(* CODESYS project vestidor.project
   Title: pl3
   Version: 0.0.0.0
   Author: ALUMNO

Project tree, tasks and I/O mapping:
  MyController : TM241CEC24R, Schneider Electric, order no. TM241CEC24R, version 4.0.6.18
      settings: OPCUA enable = True; Dummy int param for online change = 17
    application Application
      task MAST (cyclic, interval 20 ms, priority 15, watchdog 100 ms x 1) calls Main
      global variables GVL
      program Ua_control [FBD]
      OPCUASymbolConfiguration
      program Main [FBD]
      program Local_control [FBD]
    DI : Digital Inputs, Schneider Electric, version 4.0.6.18
        input  iwDI_IW0 : WORD  // IW0
        input  Application.Local_control.boolResetLocal : BOOL  // IW0.I0
        input  Application.Main.boolDeactivateStop : BOOL  // IW0.I1
        input  Application.Local_control.boolSetPosition : BOOL  // IW0.I2
        input  ibDI_IB1 : BYTE  // IB1
    DQ : Digital Outputs, Schneider Electric, version 4.0.6.18
        output Application.Main.ledLocalControl : BOOL  // QW0.Q0
        output Application.Main.ledUaControl : BOOL  // QW0.Q1
        output qbDQ_QB1 : BYTE  // QB1
        unmapped channels: QW0
    Counters : Counters, Schneider Electric, version 4.0.6.18
    Pulse_Generators : Pulse Generators, Schneider Electric, version 4.0.6.18
    Cartridge_1 : Cartridge, Schneider Electric, version 4.0.6.18
    IO_Bus : IO bus - TM3, Schneider Electric, version 4.0.6.18
    COM_Bus : COM bus, Schneider Electric, version 4.0.6.18
    Ethernet_1 : Ethernet Network, Schneider Electric, version 4.0.6.18
        settings: IPAddress = [10, 0, 0, 41]; SubnetMask = [255, 255, 0, 0]; GatewayAddress = [10, 0, 0, 1]; WebServer = TRUE; FTP Server = TRUE; SoMachine Protocol = TRUE; Modbus Server = TRUE; NetManage Protocol = TRUE; SNMP protocol = TRUE; Enable Routing = FALSE; WebVisu protocol = TRUE; DHCP Server Active = TRUE
    Serial_Line_1 : Serial line, Schneider Electric, version 4.0.6.18
      SoMachine_Network_Manager : SoMachine-Network Manager, Schneider Electric, version 4.0.0.2
    Serial_Line_2 : Serial line, Schneider Electric, version 4.0.6.18
      Modbus_Manager : Modbus Manager, Schneider Electric, version 4.0.0.2
    CAN_1 : CANopen bus, Schneider Electric, version 4.0.6.18
      CANopen_Performance : CANopen Performance, Schneider Electric, order no. 1806, version 3.0.1.24
          settings: ConfigVersion = 50659584
        Lexium_32_M : Lexium 32 M, Schneider Electric, order no. 91200, version 3.5.9.0
            settings: General Options.Optional Device = TRUE; NODEIDSAVED = 1; SDO Timeout = 1000000; Explicit Deactivate PDOs = FALSE; EXPERTSETTINGS = True; Heartbeat-Producer Time = 200; PDO 16#1400.COBID = 16#0201; PDO 16#1801.COBID = 16#C0000281; Generic COBID = '$NODEID+16#C0000280'; PDO 16#1802.COBID = 16#C0000381; Generic COBID = '$NODEID+16#C0000380'; PDO 16#1803.COBID = 16#40000481; Generic COBID = '$NODEID+16#C0000480'; Heartbeat-Consuming1.Heartbeat-Time = 300 ms; Controlword.Subindex = 16#00; Target position.Subindex = 16#00; Controlword.Subindex = 16#00; Target velocity.Subindex = 16#00; Statusword.Subindex = 16#00; Position actual value.Subindex = 16#00; Statusword.Subindex = 16#00; Velocity actual value.Subindex = 16#00; _IO_act.Index = 16#3008; _IO_act.Subindex = 16#01; _IO_act.ObjectLength = 16; _IOM1_AI11_act.Index = 16#304F; _IOM1_AI11_act.Subindex = 16#01; _IOM1_AI11_act.ObjectLength = 16; SDO List.Set Guardtime.Index = 16#100C; SDO List.Set Guardtime.Subindex = 16#00; SDO List.Set Guardtime.Value = 16#00000000; SDO List.Set Guardtime.Size = 16; SDO List.Set Guardtime.AbortIfError = FALSE; SDO List.Set Guardtime.JumpToLine = FALSE; SDO List.Set Guardtime.Line = 0; SDO List.Set Lifetime.Index = 16#100D; SDO List.Set Lifetime.Subindex = 16#00; SDO List.Set Lifetime.Value = 16#00000000; SDO List.Set Lifetime.Size = 8; SDO List.Set Lifetime.AbortIfError = FALSE;
              SDO List.Set Lifetime.JumpToLine = FALSE; SDO List.Set Lifetime.Line = 0; SDO List.Disable Emcy CobID.Index = 16#1014; SDO List.Disable Emcy CobID.Subindex = 16#00; SDO List.Disable Emcy CobID.Value = 16#80000081; SDO List.Disable Emcy CobID.Size = 32; SDO List.Disable Emcy CobID.AbortIfError = FALSE; SDO List.Disable Emcy CobID.JumpToLine = FALSE; SDO List.Disable Emcy CobID.Line = 0; SDO List.Set Emcy CobID.Index = 16#1014; SDO List.Set Emcy CobID.Subindex = 16#00; SDO List.Set Emcy CobID.Value = 16#00000081; SDO List.Set Emcy CobID.Size = 32; SDO List.Set Emcy CobID.AbortIfError = FALSE; SDO List.Set Emcy CobID.JumpToLine = FALSE; SDO List.Set Emcy CobID.Line = 0; SDO List.Set Heartbeat Consumer.Index = 16#1016; SDO List.Set Heartbeat Consumer.Subindex = 16#01; SDO List.Set Heartbeat Consumer.Value = 16#007F012C; SDO List.Set Heartbeat Consumer.Size = 32; SDO List.Set Heartbeat Consumer.AbortIfError = FALSE; SDO List.Set Heartbeat Consumer.JumpToLine = FALSE; SDO List.Set Heartbeat Consumer.Line = 0; SDO List.Set Heartbeat Consumer.Index = 16#1016; SDO List.Set Heartbeat Consumer.Subindex = 16#02; SDO List.Set Heartbeat Consumer.Value = 0; SDO List.Set Heartbeat Consumer.Size = 32; SDO List.Set Heartbeat Consumer.AbortIfError = FALSE; SDO List.Set Heartbeat Consumer.JumpToLine = FALSE; SDO List.Set Heartbeat Consumer.Line = 0; SDO List.Set Heartbeat Consumer.Index = 16#1016; SDO List.Set Heartbeat Consumer.Subindex = 16#03; SDO List.Set Heartbeat Consumer.Value = 0; SDO List.Set Heartbeat Consumer.Size = 32; SDO List.Set Heartbeat Consumer.AbortIfError = FALSE; SDO List.Set Heartbeat Consumer.JumpToLine = FALSE; SDO List.Set Heartbeat Consumer.Line = 0; SDO List.Set Heartbeat Producer.Index = 16#1017; SDO List.Set Heartbeat Producer.Subindex = 16#00; SDO List.Set Heartbeat Producer.Value = 16#000000C8;
              SDO List.Set Heartbeat Producer.Size = 16; SDO List.Set Heartbeat Producer.AbortIfError = FALSE; SDO List.Set Heartbeat Producer.JumpToLine = FALSE; SDO List.Set Heartbeat Producer.Line = 0; SDO List.Disable PDO.Index = 16#1400; SDO List.Disable PDO.Subindex = 16#01; SDO List.Disable PDO.Value = 16#80000201; SDO List.Disable PDO.Size = 32; SDO List.Disable PDO.AbortIfError = FALSE; SDO List.Disable PDO.JumpToLine = FALSE; SDO List.Disable PDO.Line = 0; SDO List.Set transmission type.Index = 16#1400; SDO List.Set transmission type.Subindex = 16#02; SDO List.Set transmission type.Value = 16#FF; SDO List.Set transmission type.Size = 8; SDO List.Set transmission type.AbortIfError = FALSE; SDO List.Set transmission type.JumpToLine = FALSE; SDO List.Set transmission type.Line = 0; SDO List.Clear pdo mapping.Index = 16#1600; SDO List.Clear pdo mapping.Subindex = 16#00; SDO List.Clear pdo mapping.Value = 16#0; SDO List.Clear pdo mapping.Size = 8; SDO List.Clear pdo mapping.AbortIfError = FALSE; SDO List.Clear pdo mapping.JumpToLine = FALSE; SDO List.Clear pdo mapping.Line = 0; SDO List.Set Mapping.Index = 16#1600; SDO List.Set Mapping.Subindex = 16#01; SDO List.Set Mapping.Value = 16#301B1F10; SDO List.Set Mapping.Size = 32; SDO List.Set Mapping.AbortIfError = FALSE; SDO List.Set Mapping.JumpToLine = FALSE; SDO List.Set Mapping.Line = 0; SDO List.Set Mapping.Index = 16#1600; SDO List.Set Mapping.Subindex = 16#02; SDO List.Set Mapping.Value = 16#301B2210; SDO List.Set Mapping.Size = 32; SDO List.Set Mapping.AbortIfError = FALSE; SDO List.Set Mapping.JumpToLine = FALSE; SDO List.Set Mapping.Line = 0; SDO List.Set Mapping.Index = 16#1600;
              SDO List.Set Mapping.Subindex = 16#03; SDO List.Set Mapping.Value = 16#301B2120; SDO List.Set Mapping.Size = 32; SDO List.Set Mapping.AbortIfError = FALSE; SDO List.Set Mapping.JumpToLine = FALSE; SDO List.Set Mapping.Line = 0; SDO List.Set number of pdos.Index = 16#1600; SDO List.Set number of pdos.Subindex = 16#00; SDO List.Set number of pdos.Value = 16#03; SDO List.Set number of pdos.Size = 8; SDO List.Set number of pdos.AbortIfError = FALSE; SDO List.Set number of pdos.JumpToLine = FALSE; SDO List.Set number of pdos.Line = 0; SDO List.Set and enable COB-ID.Index = 16#1400; SDO List.Set and enable COB-ID.Subindex = 16#01; SDO List.Set and enable COB-ID.Value = 16#00000201; SDO List.Set and enable COB-ID.Size = 32; SDO List.Set and enable COB-ID.AbortIfError = FALSE; SDO List.Set and enable COB-ID.JumpToLine = FALSE; SDO List.Set and enable COB-ID.Line = 0; SDO List.Disable PDO.Index = 16#1401; SDO List.Disable PDO.Subindex = 16#01; SDO List.Disable PDO.Value = 16#80000301; SDO List.Disable PDO.Size = 32; SDO List.Disable PDO.AbortIfError = FALSE; SDO List.Disable PDO.JumpToLine = FALSE; SDO List.Disable PDO.Line = 0; SDO List.Disable PDO.Index = 16#1402; SDO List.Disable PDO.Subindex = 16#01; SDO List.Disable PDO.Value = 16#80000401; SDO List.Disable PDO.Size = 32; SDO List.Disable PDO.AbortIfError = FALSE; SDO List.Disable PDO.JumpToLine = FALSE; SDO List.Disable PDO.Line = 0; SDO List.Disable PDO.Index = 16#1403; SDO List.Disable PDO.Subindex = 16#01; SDO List.Disable PDO.Value = 16#80000501; SDO List.Disable PDO.Size = 32; SDO List.Disable PDO.AbortIfError = FALSE; SDO List.Disable PDO.JumpToLine = FALSE;
              SDO List.Disable PDO.Line = 0; SDO List.Disable PDO.Index = 16#1800; SDO List.Disable PDO.Subindex = 16#01; SDO List.Disable PDO.Value = 16#C0000181; SDO List.Disable PDO.Size = 32; SDO List.Disable PDO.AbortIfError = FALSE; SDO List.Disable PDO.JumpToLine = FALSE; SDO List.Disable PDO.Line = 0; SDO List.Set transmission type.Index = 16#1800; SDO List.Set transmission type.Subindex = 16#02; SDO List.Set transmission type.Value = 16#FF; SDO List.Set transmission type.Size = 8; SDO List.Set transmission type.AbortIfError = FALSE; SDO List.Set transmission type.JumpToLine = FALSE; SDO List.Set transmission type.Line = 0; SDO List.Set inhibit time.Index = 16#1800; SDO List.Set inhibit time.Subindex = 16#03; SDO List.Set inhibit time.Value = 16#0064; SDO List.Set inhibit time.Size = 16; SDO List.Set inhibit time.AbortIfError = FALSE; SDO List.Set inhibit time.JumpToLine = FALSE; SDO List.Set inhibit time.Line = 0; SDO List.Set event time.Index = 16#1800; SDO List.Set event time.Subindex = 16#05; SDO List.Set event time.Value = 16#0000; SDO List.Set event time.Size = 16; SDO List.Set event time.AbortIfError = FALSE; SDO List.Set event time.JumpToLine = FALSE; SDO List.Set event time.Line = 0; SDO List.Clear pdo mapping.Index = 16#1A00; SDO List.Clear pdo mapping.Subindex = 16#00; SDO List.Clear pdo mapping.Value = 16#0; SDO List.Clear pdo mapping.Size = 8; SDO List.Clear pdo mapping.AbortIfError = FALSE; SDO List.Clear pdo mapping.JumpToLine = FALSE; SDO List.Clear pdo mapping.Line = 0; SDO List.Set Mapping.Index = 16#1A00; SDO List.Set Mapping.Subindex = 16#01; SDO List.Set Mapping.Value = 16#301B2510; SDO List.Set Mapping.Size = 32;
              SDO List.Set Mapping.AbortIfError = FALSE; SDO List.Set Mapping.JumpToLine = FALSE; SDO List.Set Mapping.Line = 0; SDO List.Set Mapping.Index = 16#1A00; SDO List.Set Mapping.Subindex = 16#02; SDO List.Set Mapping.Value = 16#301B2610; SDO List.Set Mapping.Size = 32; SDO List.Set Mapping.AbortIfError = FALSE; SDO List.Set Mapping.JumpToLine = FALSE; SDO List.Set Mapping.Line = 0; SDO List.Set Mapping.Index = 16#1A00; SDO List.Set Mapping.Subindex = 16#03; SDO List.Set Mapping.Value = 16#301B2710; SDO List.Set Mapping.Size = 32; SDO List.Set Mapping.AbortIfError = FALSE; SDO List.Set Mapping.JumpToLine = FALSE; SDO List.Set Mapping.Line = 0; SDO List.Set Mapping.Index = 16#1A00; SDO List.Set Mapping.Subindex = 16#04; SDO List.Set Mapping.Value = 16#301B2810; SDO List.Set Mapping.Size = 32; SDO List.Set Mapping.AbortIfError = FALSE; SDO List.Set Mapping.JumpToLine = FALSE; SDO List.Set Mapping.Line = 0; SDO List.Set number of pdos.Index = 16#1A00; SDO List.Set number of pdos.Subindex = 16#00; SDO List.Set number of pdos.Value = 16#04; SDO List.Set number of pdos.Size = 8; SDO List.Set number of pdos.AbortIfError = FALSE; SDO List.Set number of pdos.JumpToLine = FALSE; SDO List.Set number of pdos.Line = 0; SDO List.Set and enable COB-ID.Index = 16#1800; SDO List.Set and enable COB-ID.Subindex = 16#01; SDO List.Set and enable COB-ID.Value = 16#40000181; SDO List.Set and enable COB-ID.Size = 32; SDO List.Set and enable COB-ID.AbortIfError = FALSE; SDO List.Set and enable COB-ID.JumpToLine = FALSE; SDO List.Set and enable COB-ID.Line = 0; SDO List.Disable PDO.Index = 16#1801; SDO List.Disable PDO.Subindex = 16#01;
              SDO List.Disable PDO.Value = 16#C0000281; SDO List.Disable PDO.Size = 32; SDO List.Disable PDO.AbortIfError = FALSE; SDO List.Disable PDO.JumpToLine = FALSE; SDO List.Disable PDO.Line = 0; SDO List.Disable PDO.Index = 16#1802; SDO List.Disable PDO.Subindex = 16#01; SDO List.Disable PDO.Value = 16#C0000381; SDO List.Disable PDO.Size = 32; SDO List.Disable PDO.AbortIfError = FALSE; SDO List.Disable PDO.JumpToLine = FALSE; SDO List.Disable PDO.Line = 0; SDO List.Disable PDO.Index = 16#1803; SDO List.Disable PDO.Subindex = 16#01; SDO List.Disable PDO.Value = 16#C0000481; SDO List.Disable PDO.Size = 32; SDO List.Disable PDO.AbortIfError = FALSE; SDO List.Disable PDO.JumpToLine = FALSE; SDO List.Disable PDO.Line = 0; SDO List.Set transmission type.Index = 16#1803; SDO List.Set transmission type.Subindex = 16#02; SDO List.Set transmission type.Value = 16#FE; SDO List.Set transmission type.Size = 8; SDO List.Set transmission type.AbortIfError = FALSE; SDO List.Set transmission type.JumpToLine = FALSE; SDO List.Set transmission type.Line = 0; SDO List.Set inhibit time.Index = 16#1803; SDO List.Set inhibit time.Subindex = 16#03; SDO List.Set inhibit time.Value = 16#0000; SDO List.Set inhibit time.Size = 16; SDO List.Set inhibit time.AbortIfError = FALSE; SDO List.Set inhibit time.JumpToLine = FALSE; SDO List.Set inhibit time.Line = 0; SDO List.Set event time.Index = 16#1803; SDO List.Set event time.Subindex = 16#05; SDO List.Set event time.Value = 16#0000; SDO List.Set event time.Size = 16; SDO List.Set event time.AbortIfError = FALSE; SDO List.Set event time.JumpToLine = FALSE; SDO List.Set event time.Line = 0;
              SDO List.Clear pdo mapping.Index = 16#1A03; SDO List.Clear pdo mapping.Subindex = 16#00; SDO List.Clear pdo mapping.Value = 16#0; SDO List.Clear pdo mapping.Size = 8; SDO List.Clear pdo mapping.AbortIfError = FALSE; SDO List.Clear pdo mapping.JumpToLine = FALSE; SDO List.Clear pdo mapping.Line = 0; SDO List.Set Mapping.Index = 16#1A03; SDO List.Set Mapping.Subindex = 16#01; SDO List.Set Mapping.Value = 16#30080110; SDO List.Set Mapping.Size = 32; SDO List.Set Mapping.AbortIfError = FALSE; SDO List.Set Mapping.JumpToLine = FALSE; SDO List.Set Mapping.Line = 0; SDO List.Set Mapping.Index = 16#1A03; SDO List.Set Mapping.Subindex = 16#02; SDO List.Set Mapping.Value = 16#304F0110; SDO List.Set Mapping.Size = 32; SDO List.Set Mapping.AbortIfError = FALSE; SDO List.Set Mapping.JumpToLine = FALSE; SDO List.Set Mapping.Line = 0; SDO List.Set number of pdos.Index = 16#1A03; SDO List.Set number of pdos.Subindex = 16#00; SDO List.Set number of pdos.Value = 16#02; SDO List.Set number of pdos.Size = 8; SDO List.Set number of pdos.AbortIfError = FALSE; SDO List.Set number of pdos.JumpToLine = FALSE; SDO List.Set number of pdos.Line = 0; SDO List.Set and enable COB-ID.Index = 16#1803; SDO List.Set and enable COB-ID.Subindex = 16#01; SDO List.Set and enable COB-ID.Value = 16#40000481; SDO List.Set and enable COB-ID.Size = 32; SDO List.Set and enable COB-ID.AbortIfError = FALSE; SDO List.Set and enable COB-ID.JumpToLine = FALSE; SDO List.Set and enable COB-ID.Line = 0; SDO List.Automap SDO1.Index = 16#3041; SDO List.Automap SDO1.Subindex = 16#0B; SDO List.Automap SDO1.Value = 15; SDO List.Automap SDO1.Size = 16; SDO List.Automap SDO1.AbortIfError = FALSE;
              SDO List.Automap SDO1.JumpToLine = FALSE; SDO List.Automap SDO1.Line = 0; SDO List.Automap SDO2.Index = 16#301B; SDO List.Automap SDO2.Subindex = 16#08; SDO List.Automap SDO2.Value = 1; SDO List.Automap SDO2.Size = 16; SDO List.Automap SDO2.AbortIfError = FALSE; SDO List.Automap SDO2.JumpToLine = FALSE; SDO List.Automap SDO2.Line = 0; SDO List.Automap SDO3.Index = 16#301B; SDO List.Automap SDO3.Subindex = 16#1E; SDO List.Automap SDO3.Value = 10; SDO List.Automap SDO3.Size = 16; SDO List.Automap SDO3.AbortIfError = FALSE; SDO List.Automap SDO3.JumpToLine = FALSE; SDO List.Automap SDO3.Line = 0; ConfigVersion = 50659584
            input  Application.Local_control.boolPowerOnLocal : BOOL  // _IO_act.Bit1
            input  Application.Main.isLocal : BOOL  // _IO_act.Bit5
            input  Application.Local_control.potentiometer1 : INT  // _IOM1_AI11_act
            unmapped channels: driveModeCtrl, RefA16, RefB32, driveStat, mfStat, motionStat, driveInput, _IO_act
*)

// MyController/Application/GVL
VAR_GLOBAL
	max_vel: INT:=200;
END_VAR

// MyController/Application/Main
PROGRAM Main
VAR
	//////////////////////
	TORQUE_MAX: INT:= 300;	
	//////////////////////
	
	// Para decidir que POU correr
	isLocal: BOOL; // Asignado a PDO
	// Leds para indicarlo
	ledUaControl: BOOL; // Asginado a DQ del PLC
	ledLocalControl: BOOL; // Asignado a DQ del PLC
	// Para hacer halt en cambio de control local a Ua
	isHalt: BOOL;
	FallingEdgeLocalControl_trigg: F_TRIG;
	HaltStopLocalControlModule: MC_Halt_LXM;
	// Lectura continua del torque para parada de emergencia
	TorqueReadModule: MC_ReadActualTorque_LXM;
	actualTorque: INT;
	boolDeactivateStop: BOOL; // Asignado a DI del PLC
	HighTorqueSetReset: SR;
	isHighTorque: BOOL;
	HighTorqueStopModule: MC_Stop_LXM;	
	isStop: BOOL;
END_VAR
VAR // added by the converter: edge detectors and wires of the graphical bodies
    _w1, _w2 : BOOL;
END_VAR

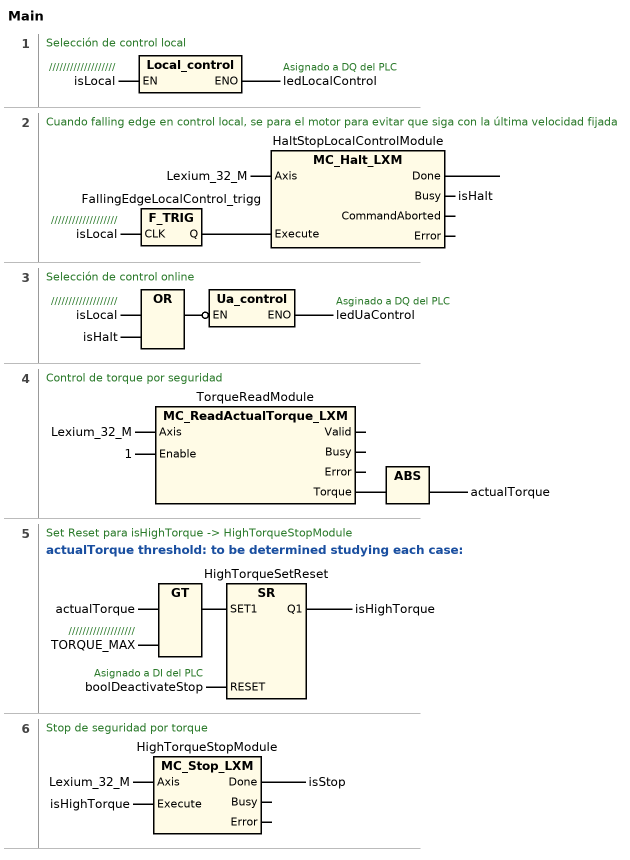
// NETWORK 1
// Selección de control local
//   isLocal: ///////////////////
//   ledLocalControl: Asignado a DQ del PLC
_w1 := isLocal;
IF _w1 THEN Local_control(); END_IF
ledLocalControl := _w1;

// NETWORK 2
// Cuando falling edge en control local, se para el motor para evitar que siga con la última velocidad fijada
//   isLocal: ///////////////////
FallingEdgeLocalControl_trigg(CLK := isLocal); // F_TRIG
HaltStopLocalControlModule(Axis := Lexium_32_M, Execute := FallingEdgeLocalControl_trigg.Q, Busy => isHalt); // MC_Halt_LXM

// NETWORK 3
// Selección de control online
//   isLocal: ///////////////////
//   ledUaControl: Asginado a DQ del PLC
_w2 := NOT (isLocal OR isHalt);
IF _w2 THEN Ua_control(); END_IF
ledUaControl := _w2;

// NETWORK 4
// Control de torque por seguridad
//   TorqueReadModule: Lectura continua del torque para parada de emergencia
TorqueReadModule(Axis := Lexium_32_M, Enable := 1); // MC_ReadActualTorque_LXM
actualTorque := ABS(TorqueReadModule.Torque);

// NETWORK 5
// Set Reset para isHighTorque -> HighTorqueStopModule
//   TORQUE_MAX: ///////////////////
//   boolDeactivateStop: Asignado a DI del PLC
// label: actualTorque threshold: to be determined studying each case
HighTorqueSetReset(SET1 := actualTorque > TORQUE_MAX, RESET := boolDeactivateStop); // SR
isHighTorque := HighTorqueSetReset.Q1;

// NETWORK 6
// Stop de seguridad por torque
HighTorqueStopModule(Axis := Lexium_32_M, Execute := isHighTorque); // MC_Stop_LXM
isStop := HighTorqueStopModule.Done;

END_PROGRAM

// MyController/Application/Local_control
PROGRAM Local_control
VAR
	//////////////////////////
	POT_MAX_VALUE: INT:=10000;
	DEAD_ZONE: INT:=1000;	
	//////////////////////////
	
	boolPowerOnLocal: BOOL;  // Asignado a PDO
	PowerOnModuleLocal: MC_Power_LXM;
	
	boolResetLocal: BOOL;	// Asignado a DI del PLC
	ResetModuleLocal: MC_Reset_LXM;
	// Control de la velocidad
	isMove: BOOL;
	potentiometer1: INT;
	isPotentiometer: BOOL;
	potentiometer2velocity: INT:=POT_MAX_VALUE/max_vel;
	MoveVelocityModuleLocal: MC_MoveVelocity_LXM;
	// Parar motor cuando entre en zona muerta
	isHaltBusy: BOOL;
	DetectFallingEdge_trigg: F_TRIG;
	HaltModuleLocal: MC_Halt_LXM;
	SetPositionModuleLocal: MC_SetPosition_LXM;
	boolSetPosition: BOOL;
END_VAR
VAR // added by the converter: edge detectors and wires of the graphical bodies
    _w1 : BOOL;
END_VAR

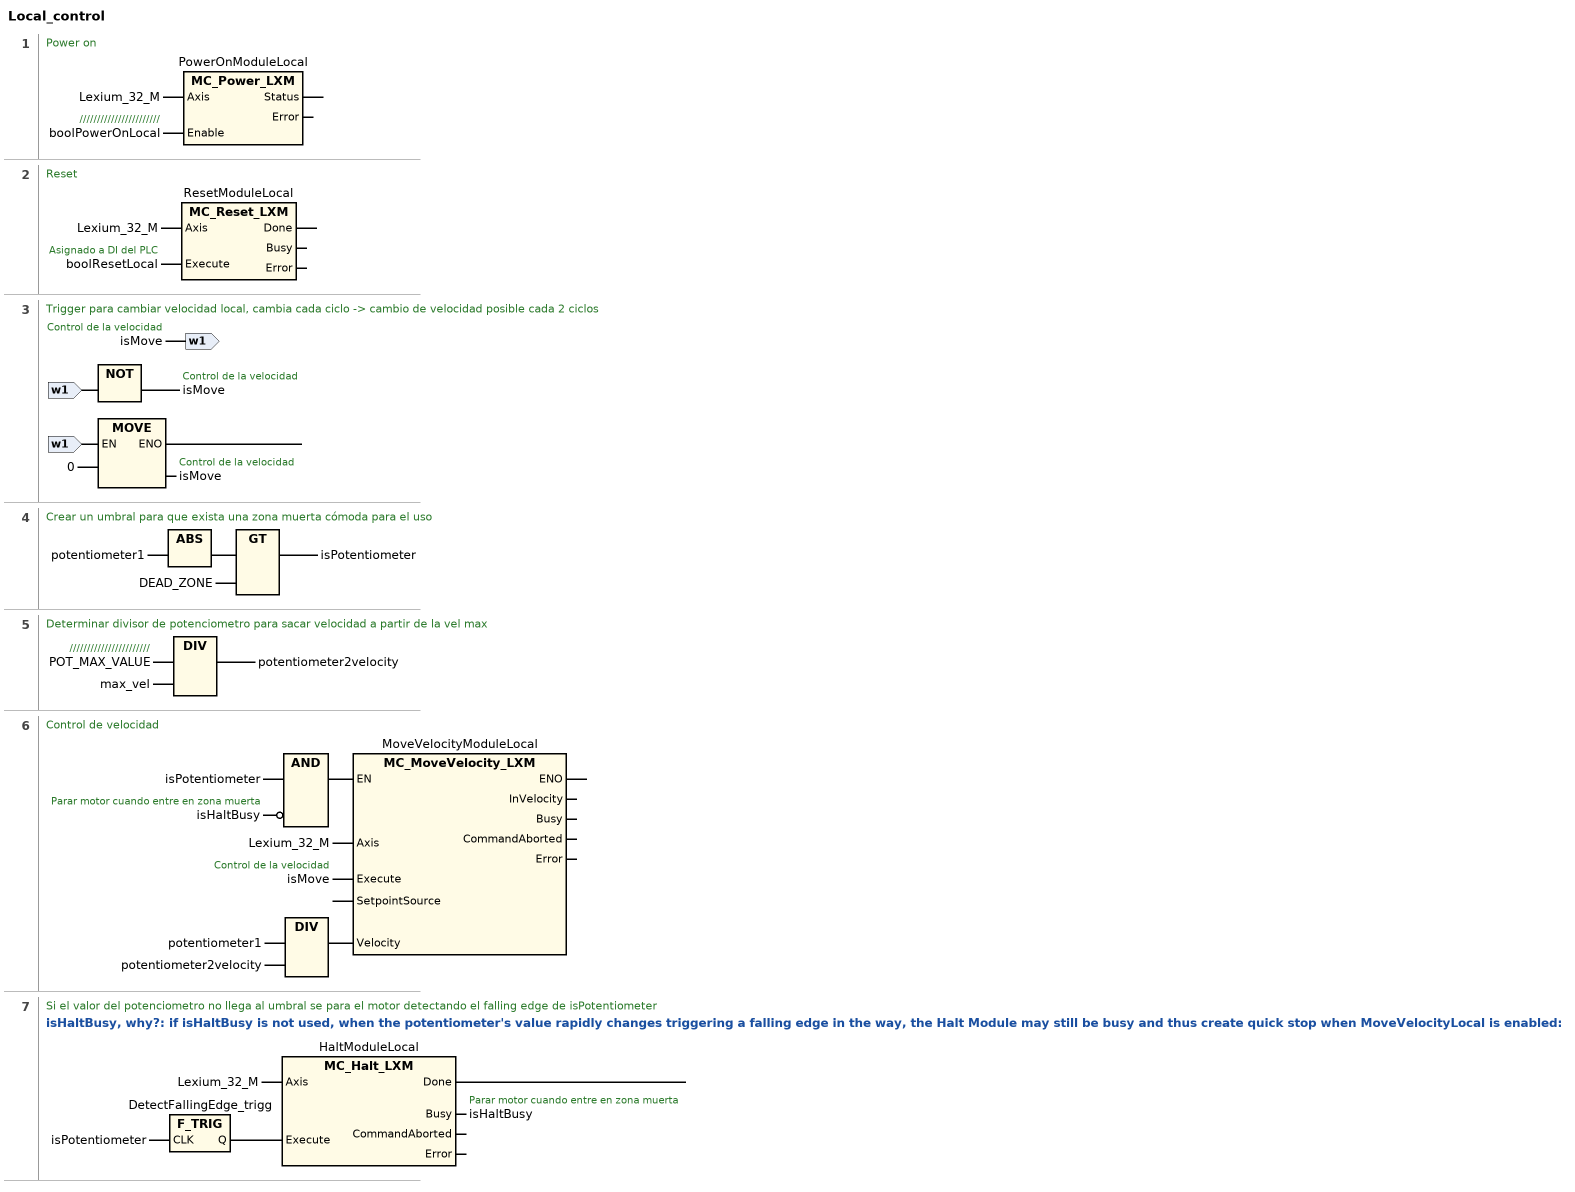
// NETWORK 1
// Power on
//   boolPowerOnLocal: ///////////////////////
PowerOnModuleLocal(Axis := Lexium_32_M, Enable := boolPowerOnLocal); // MC_Power_LXM

// NETWORK 2
// Reset
//   boolResetLocal: Asignado a DI del PLC
ResetModuleLocal(Axis := Lexium_32_M, Execute := boolResetLocal); // MC_Reset_LXM

// NETWORK 3
// Trigger para cambiar velocidad local, cambia cada ciclo -> cambio de velocidad posible cada 2 ciclos
//   isMove: Control de la velocidad
_w1 := isMove;
isMove := NOT _w1;
IF _w1 THEN isMove := 0; END_IF

// NETWORK 4
// Crear un umbral para que exista una zona muerta cómoda para el uso
isPotentiometer := ABS(potentiometer1) > DEAD_ZONE;

// NETWORK 5
// Determinar divisor de potenciometro para sacar velocidad a partir de la vel max
//   POT_MAX_VALUE: ///////////////////////
potentiometer2velocity := POT_MAX_VALUE / max_vel;

// NETWORK 6
// Control de velocidad
//   isHaltBusy: Parar motor cuando entre en zona muerta
//   isMove: Control de la velocidad
IF isPotentiometer AND NOT isHaltBusy THEN
    MoveVelocityModuleLocal(
        Axis := Lexium_32_M,
        Execute := isMove,
        Velocity := potentiometer1 / potentiometer2velocity); // MC_MoveVelocity_LXM
END_IF

// NETWORK 7
// Si el valor del potenciometro no llega al umbral se para el motor detectando el falling edge de isPotentiometer
//   isHaltBusy: Parar motor cuando entre en zona muerta
// label: isHaltBusy, why?: if isHaltBusy is not used, when the potentiometer's value rapidly changes triggering a falling edge in the way, the Halt Module may still be busy and thus create quick stop when MoveVelocityLocal is enabled
DetectFallingEdge_trigg(CLK := isPotentiometer); // F_TRIG
HaltModuleLocal(Axis := Lexium_32_M, Execute := DetectFallingEdge_trigg.Q, Busy => isHaltBusy); // MC_Halt_LXM

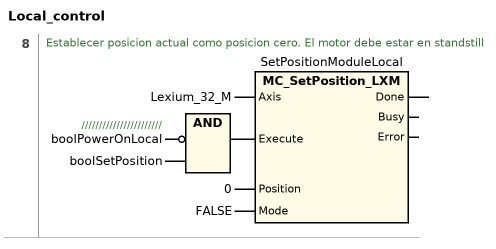
// NETWORK 8
// Establecer posicion actual como posicion cero. El motor debe estar en standstill
//   boolPowerOnLocal: ///////////////////////
SetPositionModuleLocal(
    Axis := Lexium_32_M,
    Execute := NOT boolPowerOnLocal AND boolSetPosition,
    Position := 0,
    Mode := FALSE); // MC_SetPosition_LXM

END_PROGRAM

// MyController/Application/Ua_control
PROGRAM Ua_control
VAR
	//////////////////////////
	deccDistance: INT:= 52000;
	accDistance: INT:= 16000;
	//////////////////////////
	
	PowerOnModule: MC_Power_LXM;
	boolPowerOn: BOOL;
	isPowerOn: BOOL;
	
	ResetModule: MC_Reset_LXM;
	boolReset: BOOL;
	
	HomeModule: MC_Home_LXM;
	boolHome: BOOL;
	
	// Lectura de posicion
	ReadPositionModule: MC_ReadActualPosition_LXM;
	actualPosition: DINT;
	
	//Control de movimeinto absoluto
	isMove: BOOL;
	MoveAbsoluteModule: MC_MoveAbsolute_LXM;
	selectedPosition: DINT;
	boolMoveAbsolute: BOOL;
	initPositionMoveAbsolute: DINT;
	risingEdgeMoveAbsolute_trigg: R_TRIG;
	
	//Calculo de velocidad
	velocity: INT;
	deltaSelectedPosition: INT;
	deltaInitPosition: INT;
	isDeltaInitPosition: BOOL;
	isDeltaSelectedPosition: BOOL;
	deltaMinPosition: INT;
	distance2velocity_decc: INT:=deccDistance/max_vel;
	distance2velocity_acc: INT:=accDistance/max_vel;
	
	//Change max velocity GLOBAL max_vel
	new_velocity: INT;
	boolChangeVelocity: BOOL;	
END_VAR
VAR // added by the converter: edge detectors and wires of the graphical bodies
    _w1, _w3, _w5, _w6, _w7, _w8 : BOOL;
    _w2, _w4 : INT;
END_VAR

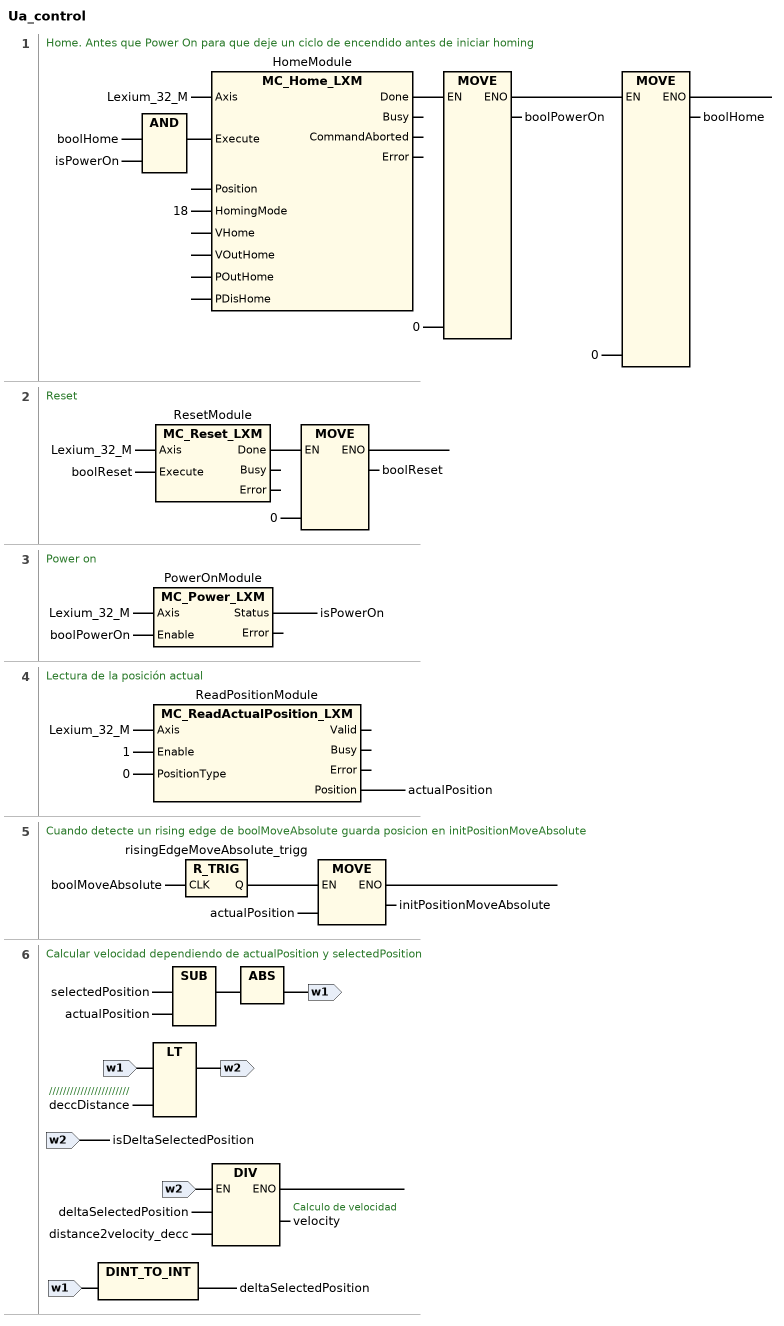
// NETWORK 1
// Home. Antes que Power On para que deje un ciclo de encendido antes de iniciar homing
HomeModule(Axis := Lexium_32_M, Execute := boolHome AND isPowerOn, HomingMode := 18); // MC_Home_LXM
_w1 := HomeModule.Done;
IF _w1 THEN boolPowerOn := 0; END_IF
IF _w1 THEN boolHome := 0; END_IF

// NETWORK 2
// Reset
ResetModule(Axis := Lexium_32_M, Execute := boolReset); // MC_Reset_LXM
IF ResetModule.Done THEN boolReset := 0; END_IF

// NETWORK 3
// Power on
//   PowerOnModule: ///////////////////////
PowerOnModule(Axis := Lexium_32_M, Enable := boolPowerOn); // MC_Power_LXM
isPowerOn := PowerOnModule.Status;

// NETWORK 4
// Lectura de la posición actual
//   ReadPositionModule: Lectura de posicion
ReadPositionModule(Axis := Lexium_32_M, Enable := 1, PositionType := 0); // MC_ReadActualPosition_LXM
actualPosition := ReadPositionModule.Position;

// NETWORK 5
// Cuando detecte un rising edge de boolMoveAbsolute guarda posicion en initPositionMoveAbsolute
risingEdgeMoveAbsolute_trigg(CLK := boolMoveAbsolute); // R_TRIG
IF risingEdgeMoveAbsolute_trigg.Q THEN initPositionMoveAbsolute := actualPosition; END_IF

// NETWORK 6
// Calcular velocidad dependiendo de actualPosition y selectedPosition
//   deccDistance: ///////////////////////
//   velocity: Calculo de velocidad
_w2 := ABS(selectedPosition - actualPosition);
_w3 := _w2 < deccDistance;
isDeltaSelectedPosition := _w3;
IF _w3 THEN velocity := deltaSelectedPosition / distance2velocity_decc; END_IF
deltaSelectedPosition := DINT_TO_INT(_w2);

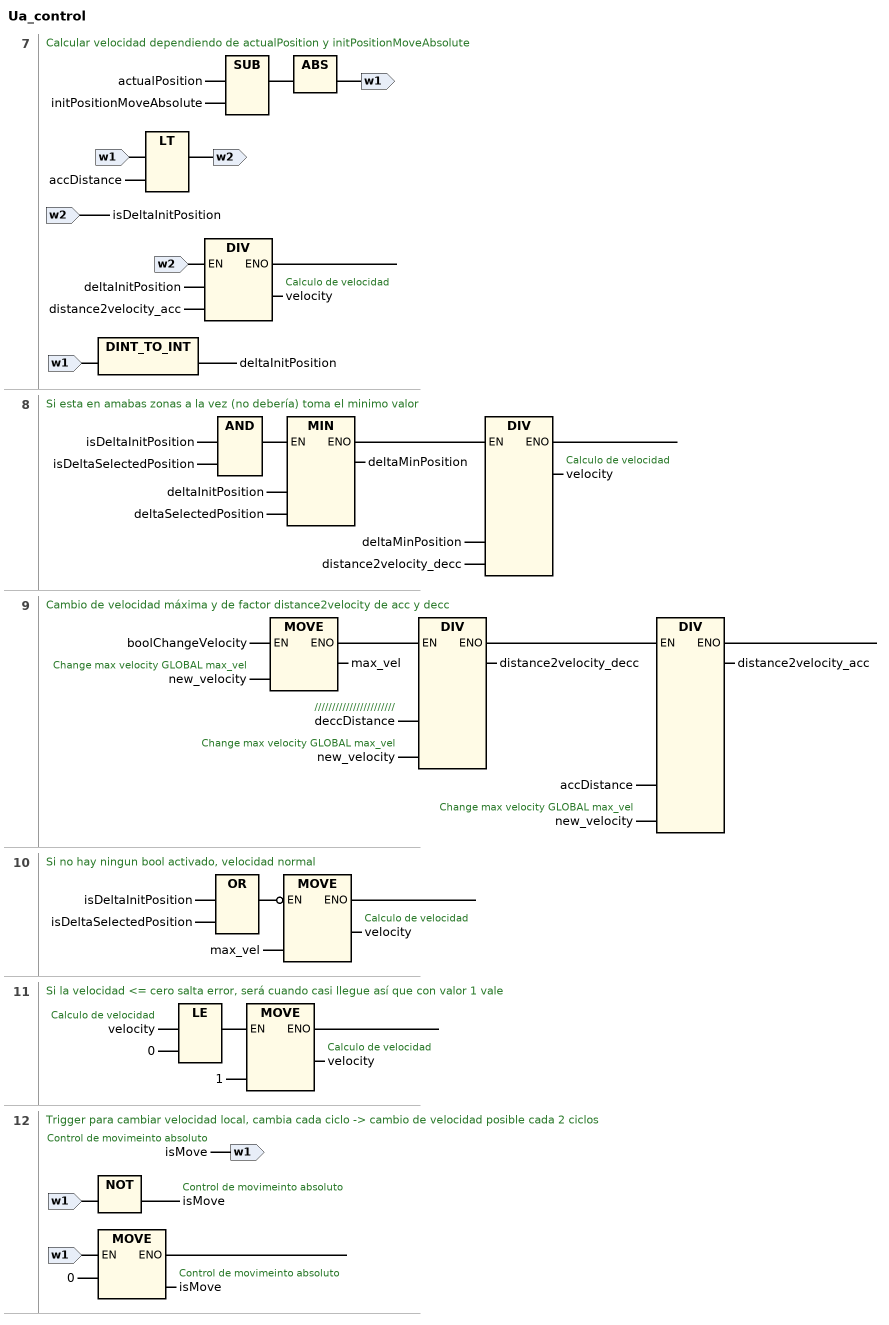
// NETWORK 7
// Calcular velocidad dependiendo de actualPosition y initPositionMoveAbsolute
//   velocity: Calculo de velocidad
_w4 := ABS(actualPosition - initPositionMoveAbsolute);
_w5 := _w4 < accDistance;
isDeltaInitPosition := _w5;
IF _w5 THEN velocity := deltaInitPosition / distance2velocity_acc; END_IF
deltaInitPosition := DINT_TO_INT(_w4);

// NETWORK 8
// Si esta en amabas zonas a la vez (no debería) toma el minimo valor
//   velocity: Calculo de velocidad
_w6 := isDeltaInitPosition AND isDeltaSelectedPosition;
IF _w6 THEN deltaMinPosition := MIN(deltaInitPosition, deltaSelectedPosition); END_IF
IF _w6 THEN velocity := deltaMinPosition / distance2velocity_decc; END_IF

// NETWORK 9
// Cambio de velocidad máxima y de factor distance2velocity de acc y decc
//   new_velocity: Change max velocity GLOBAL max_vel
//   deccDistance: ///////////////////////
_w7 := boolChangeVelocity;
IF _w7 THEN max_vel := new_velocity; END_IF
IF _w7 THEN distance2velocity_decc := deccDistance / new_velocity; END_IF
IF _w7 THEN distance2velocity_acc := accDistance / new_velocity; END_IF

// NETWORK 10
// Si no hay ningun bool activado, velocidad normal
//   velocity: Calculo de velocidad
IF NOT (isDeltaInitPosition OR isDeltaSelectedPosition) THEN velocity := max_vel; END_IF

// NETWORK 11
// Si la velocidad <= cero salta error, será cuando casi llegue así que con valor 1 vale
//   velocity: Calculo de velocidad
IF velocity <= 0 THEN velocity := 1; END_IF

// NETWORK 12
// Trigger para cambiar velocidad local, cambia cada ciclo -> cambio de velocidad posible cada 2 ciclos
//   isMove: Control de movimeinto absoluto
_w8 := isMove;
isMove := NOT _w8;
IF _w8 THEN isMove := 0; END_IF

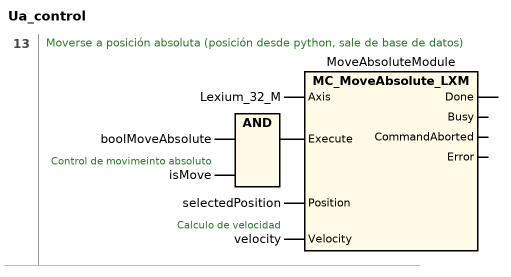
// NETWORK 13
// Moverse a posición absoluta (posición desde python, sale de base de datos)
//   isMove: Control de movimeinto absoluto
//   velocity: Calculo de velocidad
MoveAbsoluteModule(
    Axis := Lexium_32_M,
    Execute := boolMoveAbsolute AND isMove,
    Position := selectedPosition,
    Velocity := velocity); // MC_MoveAbsolute_LXM

END_PROGRAM
